{attribute 'GeneratedUsingTerminal: KL6904-0001'}
{attribute addProperty BoxType "KL6904-0001"}
{attribute addProperty Id "Channel_1AT %Q*Channel_F84AC14F0"}
{attribute addProperty CRC "2451273517"}
{attribute addProperty Size "0"}
TYPE KL_921B772D :
STRUCT
	{attribute addProperty Name "Channel_1"}
	Channel_1 : Channel_F84AC14F;
END_STRUCT
END_TYPE

(* stored: Version 1.2.0.0, ProductVersion 3.1.4024.9
   DUT KL_921B772D: Id {a3f1c5ab-6d38-4679-9d97-77d916fa3f68} *)
